Fanuc KAREL source: IO0117.KL

-- PROVISIONAL review KL for V770-1; original PC SHA256 a3296f92233a6c5f8d50fa74d9cad9873d53ab96ee1c48332be4ccc6c6d6e55c
-- Incomplete behavior may be omitted. Consult companion uncertainty JSON. Do not deploy.
PROGRAM IO0117
%NOLOCKGROUP
-- UNRESOLVED_LOCAL_POOL 5 cells at code offset 13; source declarations unknown
-- DIRECT_LOCAL_WORD_ACCESS alone does not prove INTEGER, REAL, or BOOLEAN
BEGIN
  -- UNRESOLVED_PC offsets 0-18; opcodes 2B,2C,7B
  -- UNRESOLVED_PC offsets 23-30; opcodes 9D,23
  -- UNRESOLVED_PC offsets 35-49; opcodes 2E,22,9D,33,35
  -- UNRESOLVED_PC offsets 54-61; opcodes 9D,23
  -- UNRESOLVED_PC offsets 66-77; opcodes 2E,23
  -- UNRESOLVED_PC offsets 82-91; opcodes 9D,21,1A
  -- UNRESOLVED_PC offsets 96-100; opcodes 7F
  -- UNRESOLVED_PC offsets 105-109; opcodes 27,AA
  -- UNRESOLVED_PC offsets 114-118; opcodes 7F
END IO0117
